// TIA Portal V18 export
TYPE "ServoType_UDT"
// stored: IsFailsafeCompliant false
   STRUCT
      Pos1 : Struct
         Position : Real;
         Speed : Int;
         Reached : Bool;
      END_STRUCT;
      Pos2 : Struct
         Position : Real;
         Speed : Int;
         Reached : Bool;
      END_STRUCT;
      Pos3 : Struct
         Position : Real;
         Speed : Int;
         Reached : Bool;
      END_STRUCT;
      Pos4 : Struct
         Position : Real;
         Speed : Int;
         Reached : Bool;
      END_STRUCT;
      Pos5 : Struct
         Position : Real;
         Speed : Int;
         Reached : Bool;
      END_STRUCT;
      Pos6 : Struct
         Position : Real;
         Speed : Int;
         Reached : Bool;
      END_STRUCT;
      Pos7 : Struct
         Position : Real;
         Speed : Int;
         Reached : Bool;
      END_STRUCT;
      Pos8 : Struct
         Position : Real;
         Speed : Int;
         Reached : Bool;
      END_STRUCT;
      Pos9 : Struct
         Position : Real;
         Speed : Int;
         Reached : Bool;
      END_STRUCT;
      Pos10 : Struct
         Position : Real;
         Speed : Int;
         Reached : Bool;
      END_STRUCT;
      Pos11 : Struct
         Position : Real;
         Speed : Int;
         Reached : Bool;
      END_STRUCT;
      Pos12 : Struct
         Position : Real;
         Speed : Int;
         Reached : Bool;
      END_STRUCT;
      Pos13 : Struct
         Position : Real;
         Speed : Int;
         Reached : Bool;
      END_STRUCT;
      Pos14 : Struct
         Position : Real;
         Speed : Int;
         Reached : Bool;
      END_STRUCT;
      Pos15 : Struct
         Position : Real;
         Speed : Int;
         Reached : Bool;
      END_STRUCT;
      Pos16 : Struct
         Position : Real;
         Speed : Int;
         Reached : Bool;
      END_STRUCT;
      Pos17 : Struct
         Position : Real;
         Speed : Int;
         Reached : Bool;
      END_STRUCT;
      Pos18 : Struct
         Position : Real;
         Speed : Int;
         Reached : Bool;
      END_STRUCT;
      Pos19 : Struct
         Position : Real;
         Speed : Int;
         Reached : Bool;
      END_STRUCT;
      Pos20 : Struct
         Position : Real;
         Speed : Int;
         Reached : Bool;
      END_STRUCT;
      Pos21 : Struct
         Position : Real;
         Speed : Int;
         Reached : Bool;
      END_STRUCT;
      Pos22 : Struct
         Position : Real;
         Speed : Int;
         Reached : Bool;
      END_STRUCT;
      Pos23 : Struct
         Position : Real;
         Speed : Int;
         Reached : Bool;
      END_STRUCT;
      Pos24 : Struct
         Position : Real;
         Speed : Int;
         Reached : Bool;
      END_STRUCT;
      Pos25 : Struct
         Position : Real;
         Speed : Int;
         Reached : Bool;
      END_STRUCT;
      Pos26 : Struct
         Position : Real;
         Speed : Int;
         Reached : Bool;
      END_STRUCT;
      Pos27 : Struct
         Position : Real;
         Speed : Int;
         Reached : Bool;
      END_STRUCT;
      Pos28 : Struct
         Position : Real;
         Speed : Int;
         Reached : Bool;
      END_STRUCT;
      Pos29 : Struct
         Position : Real;
         Speed : Int;
         Reached : Bool;
      END_STRUCT;
      Pos30 : Struct
         Position : Real;
         Speed : Int;
         Reached : Bool;
      END_STRUCT;
   END_STRUCT;
END_TYPE
